ABB RobotStudio station: lab2_v2.rspag

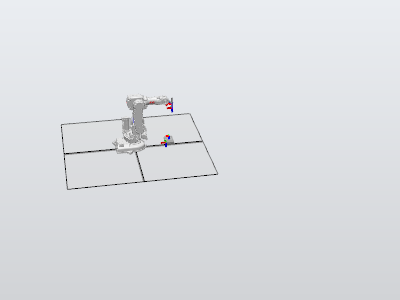
--- station ---
Station lab2_v2 (saved by RobotStudio 25.1.11167.1)
Controller IRB140_6_81
  mechanical unit ROB_1: IRB140T_6_81_C_03, 6 joints, base frame (0, 0, 0) mm
Layout (positions relative to the parent item):
  - IRB140T_6_81_C_03 [mechanism, from %ABB.RobotStudio.Models.IRB140%\IRB140T_6_81_C_G_03.rslib] at (0, 0, 0) mm; joint values [0, 0, 0, 0, 0.5236, 0] (rad or m)
  - marcador [mechanism] at (506.29, 0, 679.5) mm, rotated rx 180 ry 60 rz 180 deg
      TCP punta at (63.25, 0.5, 93.4) mm, rotated rx 0 ry 60 rz 0 deg
      links: Ensamble final v2 (1)
  - WO_LETRAS v4 [part] at (500, 0, 60) mm, rotated rx 0 ry 0 rz -90 deg, size 200 x 120 x 31 mm
Attachment: marcador is attached to IRB140T_6_81_C_03 / Link6

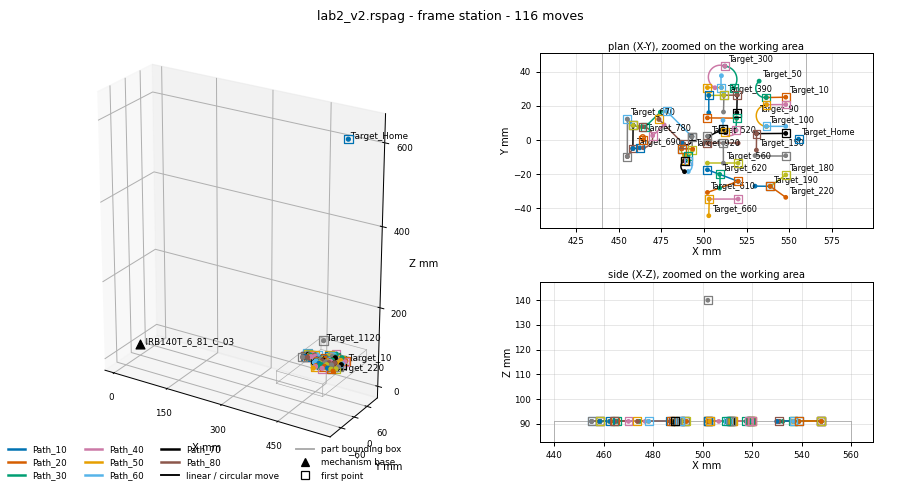
[picture p0: tool path of lab2_v2.rspag in frame station, 116 of 116 moves have a stored position in this frame; points joined in program order, loops and branches not executed]
--- Controller Data/IRB140_6_81/RAPID/TASK1/PROGMOD/CalibData.mod ---
MODULE CalibData
ENDMODULE

--- Controller Data/IRB140_6_81/RAPID/TASK1/PROGMOD/Module1.mod ---
MODULE Module1
        CONST robtarget Target_Home:=[[-115.550957906,100.5,-548.027623724],[1,0,0.000000007,0],[0,-1,0,0],[9E+09,9E+09,9E+09,9E+09,9E+09,9E+09]];
    CONST robtarget Target_10:=[[-108,125.094,-1],[1,0,0,0],[0,0,0,0],[9E+09,9E+09,9E+09,9E+09,9E+09,9E+09]];
    CONST robtarget Target_20:=[[-96.517,124.911,-1],[1,0,0,0],[0,0,0,0],[9E+09,9E+09,9E+09,9E+09,9E+09,9E+09]];
    CONST robtarget Target_30:=[[-96.579,124.938,-1],[1,0,0,0],[0,0,0,0],[9E+09,9E+09,9E+09,9E+09,9E+09,9E+09]];
    CONST robtarget Target_40:=[[-91.246,127.432,-1],[1,0,0,0],[0,0,0,0],[9E+09,9E+09,9E+09,9E+09,9E+09,9E+09]];
    CONST robtarget Target_50:=[[-92.399,134.531,-1],[1,0,0,0],[0,0,0,0],[9E+09,9E+09,9E+09,9E+09,9E+09,9E+09]];
    CONST robtarget Target_60:=[[-108,120.801,-1],[1,0,0,0],[0,0,0,0],[9E+09,9E+09,9E+09,9E+09,9E+09,9E+09]];
    CONST robtarget Target_70:=[[-96.66,120.714,-1],[1,0,0,0],[0,0,0,0],[9E+09,9E+09,9E+09,9E+09,9E+09,9E+09]];
    CONST robtarget Target_80:=[[-96.722,120.654,-1],[1,0,0,0],[0,0,0,0],[9E+09,9E+09,9E+09,9E+09,9E+09,9E+09]];
    CONST robtarget Target_90:=[[-90.707,114.263,-1],[1,0,0,0],[0,0,0,0],[9E+09,9E+09,9E+09,9E+09,9E+09,9E+09]];
    CONST robtarget Target_100:=[[-96.72,107.895,-1],[1,0,0,0],[0,0,0,0],[9E+09,9E+09,9E+09,9E+09,9E+09,9E+09]];
    CONST robtarget Target_110:=[[-96.71,108.02,-1],[1,0,0,0],[0,0,0,0],[9E+09,9E+09,9E+09,9E+09,9E+09,9E+09]];
    CONST robtarget Target_120:=[[-108,108.024,-1],[1,0,0,0],[0,0,0,0],[9E+09,9E+09,9E+09,9E+09,9E+09,9E+09]];
    CONST robtarget Target_130:=[[-108,103.869,-1],[1,0,0,0],[0,0,0,0],[9E+09,9E+09,9E+09,9E+09,9E+09,9E+09]];
    CONST robtarget Target_140:=[[-90.879,103.751,-1],[1,0,0,0],[0,0,0,0],[9E+09,9E+09,9E+09,9E+09,9E+09,9E+09]];
    CONST robtarget Target_150:=[[-90.792,94.077,-1],[1,0,0,0],[0,0,0,0],[9E+09,9E+09,9E+09,9E+09,9E+09,9E+09]];
    CONST robtarget Target_160:=[[-108,90.839,-1],[1,0,0,0],[0,0,0,0],[9E+09,9E+09,9E+09,9E+09,9E+09,9E+09]];
    CONST robtarget Target_170:=[[-90,90.839,-1],[1,0,0,0],[0,0,0,0],[9E+09,9E+09,9E+09,9E+09,9E+09,9E+09]];
    CONST robtarget Target_180:=[[-108,79.52,-1],[1,0,0,0],[0,0,0,0],[9E+09,9E+09,9E+09,9E+09,9E+09,9E+09]];
    CONST robtarget Target_190:=[[-98.899,72.871,-1],[1,0,0,0],[0,0,0,0],[9E+09,9E+09,9E+09,9E+09,9E+09,9E+09]];
    CONST robtarget Target_200:=[[-90,72.954,-1],[1,0,0,0],[0,0,0,0],[9E+09,9E+09,9E+09,9E+09,9E+09,9E+09]];
    CONST robtarget Target_210:=[[-98.899,72.871,-1],[1,0,0,0],[0,0,0,0],[9E+09,9E+09,9E+09,9E+09,9E+09,9E+09]];
    CONST robtarget Target_220:=[[-108,66.388,-1],[1,0,0,0],[0,0,0,0],[9E+09,9E+09,9E+09,9E+09,9E+09,9E+09]];
    CONST robtarget Target_230:=[[-77.51,130.536,-1],[1,0,0,0],[0,0,0,0],[9E+09,9E+09,9E+09,9E+09,9E+09,9E+09]];
    CONST robtarget Target_240:=[[-69.692,143.466,-1],[1,0,0,0],[0,0,0,0],[9E+09,9E+09,9E+09,9E+09,9E+09,9E+09]];
    CONST robtarget Target_250:=[[-67.261,130.559,-1],[1,0,0,0],[0,0,0,0],[9E+09,9E+09,9E+09,9E+09,9E+09,9E+09]];
    CONST robtarget Target_260:=[[-78.123,140.052,-1],[1,0,0,0],[0,0,0,0],[9E+09,9E+09,9E+09,9E+09,9E+09,9E+09]];
    CONST robtarget Target_270:=[[-62.805,137.7,-1],[1,0,0,0],[0,0,0,0],[9E+09,9E+09,9E+09,9E+09,9E+09,9E+09]];
    CONST robtarget Target_280:=[[-77.51,130.536,-1],[1,0,0,0],[0,0,0,0],[9E+09,9E+09,9E+09,9E+09,9E+09,9E+09]];
    CONST robtarget Target_290:=[[-78.383,139.339,-1],[1,0,0,0],[0,0,0,0],[9E+09,9E+09,9E+09,9E+09,9E+09,9E+09]];
    CONST robtarget Target_300:=[[-72.33,143.322,-1],[1,0,0,0],[0,0,0,0],[9E+09,9E+09,9E+09,9E+09,9E+09,9E+09]];
    CONST robtarget Target_310:=[[-72.33,143.322,-1],[1,0,0,0],[0,0,0,0],[9E+09,9E+09,9E+09,9E+09,9E+09,9E+09]];
    CONST robtarget Target_320:=[[-63.095,139.439,-1],[1,0,0,0],[0,0,0,0],[9E+09,9E+09,9E+09,9E+09,9E+09,9E+09]];
    CONST robtarget Target_330:=[[-66.475,130.654,-1],[1,0,0,0],[0,0,0,0],[9E+09,9E+09,9E+09,9E+09,9E+09,9E+09]];
    CONST robtarget Target_340:=[[-62.082,130.754,-1],[1,0,0,0],[0,0,0,0],[9E+09,9E+09,9E+09,9E+09,9E+09,9E+09]];
    CONST robtarget Target_350:=[[-70.29,130.75,-1],[1,0,0,0],[0,0,0,0],[9E+09,9E+09,9E+09,9E+09,9E+09,9E+09]];
    CONST robtarget Target_360:=[[-70.29,137.722,-1],[1,0,0,0],[0,0,0,0],[9E+09,9E+09,9E+09,9E+09,9E+09,9E+09]];
    CONST robtarget Target_370:=[[-79.313,116.071,-1],[1,0,0,0],[0,0,0,0],[9E+09,9E+09,9E+09,9E+09,9E+09,9E+09]];
    CONST robtarget Target_380:=[[-79.514,126.347,-1],[1,0,0,0],[0,0,0,0],[9E+09,9E+09,9E+09,9E+09,9E+09,9E+09]];
    CONST robtarget Target_390:=[[-71.742,126.235,-1],[1,0,0,0],[0,0,0,0],[9E+09,9E+09,9E+09,9E+09,9E+09,9E+09]];
    CONST robtarget Target_400:=[[-71.506,116.416,-1],[1,0,0,0],[0,0,0,0],[9E+09,9E+09,9E+09,9E+09,9E+09,9E+09]];
    CONST robtarget Target_410:=[[-71.721,126.247,-1],[1,0,0,0],[0,0,0,0],[9E+09,9E+09,9E+09,9E+09,9E+09,9E+09]];
    CONST robtarget Target_420:=[[-62.895,126.149,-1],[1,0,0,0],[0,0,0,0],[9E+09,9E+09,9E+09,9E+09,9E+09,9E+09]];
    CONST robtarget Target_430:=[[-62.874,116.003,-1],[1,0,0,0],[0,0,0,0],[9E+09,9E+09,9E+09,9E+09,9E+09,9E+09]];
    CONST robtarget Target_440:=[[-62.082,112.96,-1],[1,0,0,0],[0,0,0,0],[9E+09,9E+09,9E+09,9E+09,9E+09,9E+09]];
    CONST robtarget Target_450:=[[-79.192,112.835,-1],[1,0,0,0],[0,0,0,0],[9E+09,9E+09,9E+09,9E+09,9E+09,9E+09]];
    CONST robtarget Target_460:=[[-78.805,105.664,-1],[1,0,0,0],[0,0,0,0],[9E+09,9E+09,9E+09,9E+09,9E+09,9E+09]];
    CONST robtarget Target_470:=[[-75.79,102.587,-1],[1,0,0,0],[0,0,0,0],[9E+09,9E+09,9E+09,9E+09,9E+09,9E+09]];
    CONST robtarget Target_480:=[[-72.357,104.51,-1],[1,0,0,0],[0,0,0,0],[9E+09,9E+09,9E+09,9E+09,9E+09,9E+09]];
    CONST robtarget Target_490:=[[-71.207,106.55,-1],[1,0,0,0],[0,0,0,0],[9E+09,9E+09,9E+09,9E+09,9E+09,9E+09]];
    CONST robtarget Target_500:=[[-71.216,111.54,-1],[1,0,0,0],[0,0,0,0],[9E+09,9E+09,9E+09,9E+09,9E+09,9E+09]];
    CONST robtarget Target_510:=[[-71.224,106.472,-1],[1,0,0,0],[0,0,0,0],[9E+09,9E+09,9E+09,9E+09,9E+09,9E+09]];
    CONST robtarget Target_520:=[[-62.667,102.098,-1],[1,0,0,0],[0,0,0,0],[9E+09,9E+09,9E+09,9E+09,9E+09,9E+09]];
    CONST robtarget Target_530:=[[-62.082,98.14,-1],[1,0,0,0],[0,0,0,0],[9E+09,9E+09,9E+09,9E+09,9E+09,9E+09]];
    CONST robtarget Target_540:=[[-80.082,98.14,-1],[1,0,0,0],[0,0,0,0],[9E+09,9E+09,9E+09,9E+09,9E+09,9E+09]];
    CONST robtarget Target_550:=[[-71.397,98.148,-1],[1,0,0,0],[0,0,0,0],[9E+09,9E+09,9E+09,9E+09,9E+09,9E+09]];
    CONST robtarget Target_560:=[[-71.446,86.432,-1],[1,0,0,0],[0,0,0,0],[9E+09,9E+09,9E+09,9E+09,9E+09,9E+09]];
    CONST robtarget Target_570:=[[-80.082,86.454,-1],[1,0,0,0],[0,0,0,0],[9E+09,9E+09,9E+09,9E+09,9E+09,9E+09]];
    CONST robtarget Target_580:=[[-62.082,86.454,-1],[1,0,0,0],[0,0,0,0],[9E+09,9E+09,9E+09,9E+09,9E+09,9E+09]];
    CONST robtarget Target_590:=[[-62.082,82.562,-1],[1,0,0,0],[0,0,0,0],[9E+09,9E+09,9E+09,9E+09,9E+09,9E+09]];
    CONST robtarget Target_600:=[[-80.082,75.79,-1],[1,0,0,0],[0,0,0,0],[9E+09,9E+09,9E+09,9E+09,9E+09,9E+09]];
    CONST robtarget Target_610:=[[-62.082,69.258,-1],[1,0,0,0],[0,0,0,0],[9E+09,9E+09,9E+09,9E+09,9E+09,9E+09]];
    CONST robtarget Target_620:=[[-69.26,79.86,-1],[1,0,0,0],[0,0,0,0],[9E+09,9E+09,9E+09,9E+09,9E+09,9E+09]];
    CONST robtarget Target_630:=[[-69.26,71.805,-1],[1,0,0,0],[0,0,0,0],[9E+09,9E+09,9E+09,9E+09,9E+09,9E+09]];
    CONST robtarget Target_640:=[[-80.082,65.389,-1],[1,0,0,0],[0,0,0,0],[9E+09,9E+09,9E+09,9E+09,9E+09,9E+09]];
    CONST robtarget Target_650:=[[-63.123,65.37,-1],[1,0,0,0],[0,0,0,0],[9E+09,9E+09,9E+09,9E+09,9E+09,9E+09]];
    CONST robtarget Target_660:=[[-62.874,55.597,-1],[1,0,0,0],[0,0,0,0],[9E+09,9E+09,9E+09,9E+09,9E+09,9E+09]];
    CONST robtarget Target_670:=[[-15.067,112.238,-1],[1,0,0,0],[0,0,0,0],[9E+09,9E+09,9E+09,9E+09,9E+09,9E+09]];
    CONST robtarget Target_680:=[[-18.49,108.612,-1],[1,0,0,0],[0,0,0,0],[9E+09,9E+09,9E+09,9E+09,9E+09,9E+09]];
    CONST robtarget Target_690:=[[-18.364,95.026,-1],[1,0,0,0],[0,0,0,0],[9E+09,9E+09,9E+09,9E+09,9E+09,9E+09]];
    CONST robtarget Target_700:=[[-15.102,90.307,-1],[1,0,0,0],[0,0,0,0],[9E+09,9E+09,9E+09,9E+09,9E+09,9E+09]];
    CONST robtarget Target_710:=[[-15.158,112.207,-1],[1,0,0,0],[0,0,0,0],[9E+09,9E+09,9E+09,9E+09,9E+09,9E+09]];
    CONST robtarget Target_720:=[[-18.49,108.612,-1],[1,0,0,0],[0,0,0,0],[9E+09,9E+09,9E+09,9E+09,9E+09,9E+09]];
    CONST robtarget Target_730:=[[-22.178,107.545,-1],[1,0,0,0],[0,0,0,0],[9E+09,9E+09,9E+09,9E+09,9E+09,9E+09]];
    CONST robtarget Target_740:=[[-29.789,101.463,-1],[1,0,0,0],[0,0,0,0],[9E+09,9E+09,9E+09,9E+09,9E+09,9E+09]];
    CONST robtarget Target_750:=[[-22.386,95.374,-1],[1,0,0,0],[0,0,0,0],[9E+09,9E+09,9E+09,9E+09,9E+09,9E+09]];
    CONST robtarget Target_760:=[[-18.397,95.013,-1],[1,0,0,0],[0,0,0,0],[9E+09,9E+09,9E+09,9E+09,9E+09,9E+09]];
    CONST robtarget Target_770:=[[-24.444,100.113,-1],[1,0,0,0],[0,0,0,0],[9E+09,9E+09,9E+09,9E+09,9E+09,9E+09]];
    CONST robtarget Target_780:=[[-24.359,103.047,-1],[1,0,0,0],[0,0,0,0],[9E+09,9E+09,9E+09,9E+09,9E+09,9E+09]];
    CONST robtarget Target_790:=[[-24.554,100.141,-1],[1,0,0,0],[0,0,0,0],[9E+09,9E+09,9E+09,9E+09,9E+09,9E+09]];
    CONST robtarget Target_800:=[[-25.496,107.635,-1],[1,0,0,0],[0,0,0,0],[9E+09,9E+09,9E+09,9E+09,9E+09,9E+09]];
    CONST robtarget Target_810:=[[-34.48,116.37,-1],[1,0,0,0],[0,0,0,0],[9E+09,9E+09,9E+09,9E+09,9E+09,9E+09]];
    CONST robtarget Target_820:=[[-29.986,102.575,-1],[1,0,0,0],[0,0,0,0],[9E+09,9E+09,9E+09,9E+09,9E+09,9E+09]];
    CONST robtarget Target_830:=[[-36.719,108.862,-1],[1,0,0,0],[0,0,0,0],[9E+09,9E+09,9E+09,9E+09,9E+09,9E+09]];
    CONST robtarget Target_840:=[[-33.544,112.115,-1],[1,0,0,0],[0,0,0,0],[9E+09,9E+09,9E+09,9E+09,9E+09,9E+09]];
    CONST robtarget Target_850:=[[-34.336,116.216,-1],[1,0,0,0],[0,0,0,0],[9E+09,9E+09,9E+09,9E+09,9E+09,9E+09]];
    CONST robtarget Target_860:=[[-38.148,116.925,-1],[1,0,0,0],[0,0,0,0],[9E+09,9E+09,9E+09,9E+09,9E+09,9E+09]];
    CONST robtarget Target_870:=[[-52.946,102.081,-1],[1,0,0,0],[0,0,0,0],[9E+09,9E+09,9E+09,9E+09,9E+09,9E+09]];
    CONST robtarget Target_880:=[[-52.107,98.145,-1],[1,0,0,0],[0,0,0,0],[9E+09,9E+09,9E+09,9E+09,9E+09,9E+09]];
    CONST robtarget Target_890:=[[-48.099,97.619,-1],[1,0,0,0],[0,0,0,0],[9E+09,9E+09,9E+09,9E+09,9E+09,9E+09]];
    CONST robtarget Target_900:=[[-33.658,112.146,-1],[1,0,0,0],[0,0,0,0],[9E+09,9E+09,9E+09,9E+09,9E+09,9E+09]];
    CONST robtarget Target_910:=[[-52.993,101.964,-1],[1,0,0,0],[0,0,0,0],[9E+09,9E+09,9E+09,9E+09,9E+09,9E+09]];
    CONST robtarget Target_920:=[[-53.234,94.103,-1],[1,0,0,0],[0,0,0,0],[9E+09,9E+09,9E+09,9E+09,9E+09,9E+09]];
    CONST robtarget Target_930:=[[-50.381,90.681,-1],[1,0,0,0],[0,0,0,0],[9E+09,9E+09,9E+09,9E+09,9E+09,9E+09]];
    CONST robtarget Target_940:=[[-46.922,94.871,-1],[1,0,0,0],[0,0,0,0],[9E+09,9E+09,9E+09,9E+09,9E+09,9E+09]];
    CONST robtarget Target_950:=[[-47.013,98.691,-1],[1,0,0,0],[0,0,0,0],[9E+09,9E+09,9E+09,9E+09,9E+09,9E+09]];
    CONST robtarget Target_960:=[[-47.015,94.837,-1],[1,0,0,0],[0,0,0,0],[9E+09,9E+09,9E+09,9E+09,9E+09,9E+09]];
    CONST robtarget Target_970:=[[-53.429,94.778,-1],[1,0,0,0],[0,0,0,0],[9E+09,9E+09,9E+09,9E+09,9E+09,9E+09]];
    CONST robtarget Target_980:=[[-50.711,90.745,-1],[1,0,0,0],[0,0,0,0],[9E+09,9E+09,9E+09,9E+09,9E+09,9E+09]];
    CONST robtarget Target_990:=[[-50.919,87.918,-1],[1,0,0,0],[0,0,0,0],[9E+09,9E+09,9E+09,9E+09,9E+09,9E+09]];
    CONST robtarget Target_1000:=[[-49.871,86.938,-1],[1,0,0,0],[0,0,0,0],[9E+09,9E+09,9E+09,9E+09,9E+09,9E+09]];
    CONST robtarget Target_1010:=[[-48.634,87.988,-1],[1,0,0,0],[0,0,0,0],[9E+09,9E+09,9E+09,9E+09,9E+09,9E+09]];
    CONST robtarget Target_1020:=[[-48.643,90.985,-1],[1,0,0,0],[0,0,0,0],[9E+09,9E+09,9E+09,9E+09,9E+09,9E+09]];
    CONST robtarget Target_1030:=[[-50.973,87.895,-1],[1,0,0,0],[0,0,0,0],[9E+09,9E+09,9E+09,9E+09,9E+09,9E+09]];
    CONST robtarget Target_1040:=[[-53.036,84.502,-1],[1,0,0,0],[0,0,0,0],[9E+09,9E+09,9E+09,9E+09,9E+09,9E+09]];
    CONST robtarget Target_1050:=[[-50.844,81.528,-1],[1,0,0,0],[0,0,0,0],[9E+09,9E+09,9E+09,9E+09,9E+09,9E+09]];
    CONST robtarget Target_1060:=[[-48.691,87.835,-1],[1,0,0,0],[0,0,0,0],[9E+09,9E+09,9E+09,9E+09,9E+09,9E+09]];
    CONST robtarget Target_1070:=[[-46.541,84.777,-1],[1,0,0,0],[0,0,0,0],[9E+09,9E+09,9E+09,9E+09,9E+09,9E+09]];
    CONST robtarget Target_1080:=[[-48.635,81.464,0],[1,0,0,0],[0,0,0,0],[9E+09,9E+09,9E+09,9E+09,9E+09,9E+09]];
    CONST robtarget Target_1090:=[[-24.027,107.791,-1],[1,0,0,0],[0,0,0,0],[9E+09,9E+09,9E+09,9E+09,9E+09,9E+09]];
    CONST robtarget Target_1100:=[[-29.971,101.827,-1],[1,0,0,0],[0,0,0,0],[9E+09,9E+09,9E+09,9E+09,9E+09,9E+09]];
    CONST robtarget Target_1110:=[[-24.506,95.448,-1],[1,0,0,0],[0,0,0,0],[9E+09,9E+09,9E+09,9E+09,9E+09,9E+09]];
    CONST robtarget Target_1120:=[[-62.082,102.239,-50],[1,0,0,0],[0,0,0,0],[9E+09,9E+09,9E+09,9E+09,9E+09,9E+09]];
    PERS tooldata punta:=[TRUE,[[63.248,0.5,93.396],[0.866025404,0,0.5,0]],[1,[0,0,1],[1,0,0,0],0,0,0]];
    TASK PERS wobjdata Workobject_2:=[FALSE,TRUE,"",[[0,0,60],[1,0,0,0]],[[440,-100,30],[0,0,1,0]]];
!***********************************************************
    !
    ! M?dulo:  Module1
    !
    ! Descripción:
    !   <Introduzca la descripción aquí>
    !
    ! Autor: MacBook Air
    !
    ! Versión: 1.0
    !
    !***********************************************************


    !***********************************************************
    !
    ! Procedimiento Main
    !
    !   Este es el punto de entrada de su programa
    !
    !***********************************************************
    PROC main()
        Path_10;
        Path_600;
        Path_20;
        Path_30;
        Path_600;
        Path_40;
        Path_50;
        Path_60;
        Path_600;
        Path_70;
        Path_80;
        Path_600;
        Path_90;
        Path_600;
        Path_100;
        Path_110;
        Path_120;
        Path_600;
        Path_130;
        Path_140;
        Path_150;
        Path_160;
        Path_600;
        Path_170;
        Path_180;
        Path_190;
        Path_200;
        Path_210;
        Path_600;
        Path_220;
        Path_230;
        Path_240;
        Path_250;
        Path_260;
        Path_270;
        Path_600;
        Path_280;
        Path_290;
        Path_300;
        Path_600;
        Path_310;
        Path_320;
        Path_330;
        Path_600;
        Path_340;
        Path_350;
        Path_600;
        Path_360;
        Path_370;
        Path_380;
        Path_390;
        Path_600;
        Path_400;
        Path_600;
        Path_420;
        Path_600;
        Path_440;
        Path_600;
        Path_450;
        Path_600;
        Path_460;
        Path_470;
        Path_480;
        Path_490;
        Path_600;
        Path_500;
        Path_510;
        Path_520;
        Path_600;
        Path_530;
        Path_600;
        Path_540;
        Path_550;
        Path_560;
        Path_600;
        Path_570;
        Path_580;
        Path_600;
        Path_590;
        Path_600;
        Path_10;



    ENDPROC
    PROC Path_10()
        MoveJ Target_Home,v100,z10,punta\WObj:=Workobject_2;
    ENDPROC
    PROC Path_20()
        MoveJ Target_10,v100,z10,punta\WObj:=Workobject_2;
        MoveL Target_20,v100,z10,punta\WObj:=Workobject_2;
    ENDPROC
    PROC Path_30()
        MoveJ Target_30,v100,z10,punta\WObj:=Workobject_2;
        MoveC Target_40,Target_50,v100,z10,punta\WObj:=Workobject_2;
    ENDPROC
    PROC Path_40()
        MoveJ Target_60,v100,z10,punta\WObj:=Workobject_2;
        MoveL Target_70,v100,z10,punta\WObj:=Workobject_2;
    ENDPROC
    PROC Path_50()
        MoveJ Target_80,v100,z10,punta\WObj:=Workobject_2;
        MoveC Target_90,Target_100,v1000,z100,punta\WObj:=Workobject_2;
    ENDPROC
    PROC Path_60()
        MoveJ Target_110,v100,z10,punta\WObj:=Workobject_2;
        MoveL Target_120,v100,z10,punta\WObj:=Workobject_2;
    ENDPROC
    PROC Path_70()
        MoveJ Target_130,v100,z10,punta\WObj:=Workobject_2;
        MoveL Target_140,v100,z10,punta\WObj:=Workobject_2;
    ENDPROC
    PROC Path_80()
        MoveJ Target_140,v100,z10,punta\WObj:=Workobject_2;
        MoveL Target_150,v100,z10,punta\WObj:=Workobject_2;
    ENDPROC
    PROC Path_90()
        MoveJ Target_160,v100,z10,punta\WObj:=Workobject_2;
        MoveL Target_170,v100,z10,punta\WObj:=Workobject_2;
    ENDPROC
    PROC Path_100()
        MoveJ Target_180,v100,z10,punta\WObj:=Workobject_2;
        MoveL Target_190,v100,z10,punta\WObj:=Workobject_2;
    ENDPROC
    PROC Path_110()
        MoveJ Target_190,v100,z10,punta\WObj:=Workobject_2;
        MoveL Target_200,v100,z10,punta\WObj:=Workobject_2;
    ENDPROC
    PROC Path_120()
        MoveJ Target_210,v100,z10,punta\WObj:=Workobject_2;
        MoveL Target_220,v100,z10,punta\WObj:=Workobject_2;
    ENDPROC
    PROC Path_130()
        MoveJ Target_280,v100,z10,punta\WObj:=Workobject_2;
        MoveC Target_290,Target_300,v100,z10,punta\WObj:=Workobject_2;
    ENDPROC
    PROC Path_140()
        MoveJ Target_310,v100,z10,punta\WObj:=Workobject_2;
        MoveC Target_320,Target_330,v100,z10,punta\WObj:=Workobject_2;

    ENDPROC
    PROC Path_150()
        MoveJ Target_340,v100,z10,punta\WObj:=Workobject_2;
        MoveL Target_350,v100,z10,punta\WObj:=Workobject_2;
    ENDPROC
    PROC Path_160()
        MoveJ Target_350,v100,z10,punta\WObj:=Workobject_2;
        MoveL Target_360,v100,z10,punta\WObj:=Workobject_2;
    ENDPROC
    PROC Path_170()
        MoveJ Target_370,v100,z10,punta\WObj:=Workobject_2;
        MoveL Target_380,v100,z10,punta\WObj:=Workobject_2;
    ENDPROC
    PROC Path_180()
        MoveJ Target_380,v100,z10,punta\WObj:=Workobject_2;
        MoveL Target_390,v100,z10,punta\WObj:=Workobject_2;
    ENDPROC
    PROC Path_190()
        MoveJ Target_390,v100,z10,punta\WObj:=Workobject_2;
        MoveL Target_400,v100,z10,punta\WObj:=Workobject_2;
    ENDPROC
    PROC Path_200()
        MoveJ Target_410,v100,z10,punta\WObj:=Workobject_2;
        MoveL Target_420,v100,z10,punta\WObj:=Workobject_2;
    ENDPROC
    PROC Path_210()
        MoveJ Target_420,v100,z10,punta\WObj:=Workobject_2;
        MoveL Target_430,v100,z10,punta\WObj:=Workobject_2;
    ENDPROC
    PROC Path_220()
        MoveJ Target_440,v100,z10,punta\WObj:=Workobject_2;
        MoveL Target_450,v100,z10,punta\WObj:=Workobject_2;
    ENDPROC
    PROC Path_230()
        MoveJ Target_450,v100,z10,punta\WObj:=Workobject_2;
        MoveL Target_460,v100,z10,punta\WObj:=Workobject_2;
    ENDPROC
    PROC Path_240()
        MoveJ Target_460,v100,z10,punta\WObj:=Workobject_2;
        MoveC Target_470,Target_480,v100,z10,punta\WObj:=Workobject_2;

    ENDPROC
    PROC Path_250()
        MoveJ Target_480,v100,z10,punta\WObj:=Workobject_2;
        MoveL Target_490,v100,z10,punta\WObj:=Workobject_2;
    ENDPROC
    PROC Path_260()
        MoveJ Target_490,v100,z10,punta\WObj:=Workobject_2;
        MoveL Target_500,v100,z10,punta\WObj:=Workobject_2;
    ENDPROC
    PROC Path_270()
        MoveJ Target_510,v100,z10,punta\WObj:=Workobject_2;
        MoveL Target_520,v100,z10,punta\WObj:=Workobject_2;
    ENDPROC
    PROC Path_280()
        MoveJ Target_530,v100,z10,punta\WObj:=Workobject_2;
        MoveL Target_540,v100,z10,punta\WObj:=Workobject_2;
    ENDPROC
    PROC Path_290()
        MoveJ Target_550,v100,z10,punta\WObj:=Workobject_2;
        MoveL Target_560,v100,z10,punta\WObj:=Workobject_2;
    ENDPROC
    PROC Path_300()
        MoveJ Target_570,v100,z10,punta\WObj:=Workobject_2;
        MoveL Target_580,v100,z10,punta\WObj:=Workobject_2;
    ENDPROC
    PROC Path_310()
        MoveJ Target_590,v100,z10,punta\WObj:=Workobject_2;
        MoveL Target_600,v100,z10,punta\WObj:=Workobject_2;
    ENDPROC
    PROC Path_320()
        MoveJ Target_600,v100,z10,punta\WObj:=Workobject_2;
        MoveL Target_610,v100,z10,punta\WObj:=Workobject_2;
    ENDPROC
    PROC Path_330()
        MoveJ Target_620,v100,z10,punta\WObj:=Workobject_2;
        MoveL Target_630,v100,z10,punta\WObj:=Workobject_2;
    ENDPROC
    PROC Path_340()
        MoveJ Target_640,v100,z10,punta\WObj:=Workobject_2;
        MoveL Target_650,v100,z10,punta\WObj:=Workobject_2;
    ENDPROC
    PROC Path_350()
        MoveJ Target_650,v100,z10,punta\WObj:=Workobject_2;
        MoveL Target_660,v100,z10,punta\WObj:=Workobject_2;
    ENDPROC
    PROC Path_360()
        MoveJ Target_670,v100,z10,punta\WObj:=Workobject_2;
        MoveL Target_680,v100,z10,punta\WObj:=Workobject_2;
    ENDPROC
    PROC Path_370()
        MoveJ Target_680,v100,z10,punta\WObj:=Workobject_2;
        MoveL Target_690,v100,z10,punta\WObj:=Workobject_2;
    ENDPROC
    PROC Path_380()
        MoveJ Target_690,v100,z10,punta\WObj:=Workobject_2;
        MoveL Target_700,v100,z10,punta\WObj:=Workobject_2;
    ENDPROC
    PROC Path_390()
        MoveJ Target_700,v1000,z10,punta\WObj:=Workobject_2;
        MoveL Target_710,v1000,z10,punta\WObj:=Workobject_2;
    ENDPROC
    PROC Path_400()
        MoveJ Target_720,v100,z10,punta\WObj:=Workobject_2;
        MoveL Target_730,v100,z10,punta\WObj:=Workobject_2;
    ENDPROC

    PROC Path_420()
        MoveJ Target_750,v100,z10,punta\WObj:=Workobject_2;
        MoveL Target_760,v100,z10,punta\WObj:=Workobject_2;
    ENDPROC
    PROC Path_430()
        MoveJ Target_770,v100,z10,punta\WObj:=Workobject_2;
        MoveC Target_780,Target_790,v100,z10,punta\WObj:=Workobject_2;

    ENDPROC
    PROC Path_440()
        MoveJ Target_800,v100,z10,punta\WObj:=Workobject_2;
        MoveL Target_810,v100,z10,punta\WObj:=Workobject_2;
    ENDPROC
    PROC Path_450()
        MoveJ Target_820,v100,z10,punta\WObj:=Workobject_2;
        MoveL Target_830,v100,z10,punta\WObj:=Workobject_2;
    ENDPROC
    PROC Path_460()
        MoveJ Target_840,v100,z10,punta\WObj:=Workobject_2;
        MoveC Target_850,Target_860,v100,z10,punta\WObj:=Workobject_2;
    ENDPROC
    PROC Path_470()
        MoveJ Target_860,v100,z10,punta\WObj:=Workobject_2;
        MoveL Target_870,v100,z10,punta\WObj:=Workobject_2;
    ENDPROC
    PROC Path_480()
        MoveJ Target_870,v100,z10,punta\WObj:=Workobject_2;
        MoveC Target_880,Target_890,v100,z10,punta\WObj:=Workobject_2;
    ENDPROC
    PROC Path_490()
        MoveJ Target_890,v100,z10,punta\WObj:=Workobject_2;
        MoveL Target_900,v100,z10,punta\WObj:=Workobject_2;
    ENDPROC
    PROC Path_500()
        MoveJ Target_910,v100,z10,punta\WObj:=Workobject_2;
        MoveL Target_920,v100,z10,punta\WObj:=Workobject_2;
    ENDPROC
    PROC Path_510()
        MoveJ Target_920,v100,z10,punta\WObj:=Workobject_2;
        MoveC Target_930,Target_940,v100,z10,punta\WObj:=Workobject_2;
    ENDPROC
    PROC Path_520()
        MoveJ Target_940,v100,z10,punta\WObj:=Workobject_2;
        MoveL Target_950,v100,z10,punta\WObj:=Workobject_2;
    ENDPROC
    PROC Path_530()
        MoveJ Target_960,v100,z10,punta\WObj:=Workobject_2;
        MoveL Target_970,v100,z10,punta\WObj:=Workobject_2;
    ENDPROC
    PROC Path_540()
        MoveJ Target_980,v100,z10,punta\WObj:=Workobject_2;
        MoveL Target_990,v100,z10,punta\WObj:=Workobject_2;
    ENDPROC
    PROC Path_550()
        MoveJ Target_990,v100,z10,punta\WObj:=Workobject_2;
        MoveC Target_1000,Target_1010,v100,z10,punta\WObj:=Workobject_2;

    ENDPROC
    PROC Path_560()
        MoveJ Target_1010,v100,z10,punta\WObj:=Workobject_2;
        MoveL Target_1020,v100,z10,punta\WObj:=Workobject_2;
    ENDPROC
    PROC Path_570()
        MoveJ Target_1030,v100,z10,punta\WObj:=Workobject_2;
        MoveC Target_1040,Target_1050,v100,z10,punta\WObj:=Workobject_2;

    ENDPROC
    PROC Path_580()
        MoveJ Target_1060,v100,z10,punta\WObj:=Workobject_2;
        MoveC Target_1070,Target_1080,v100,z10,punta\WObj:=Workobject_2;

    ENDPROC
    PROC Path_590()
        MoveJ Target_1090,v100,z10,punta\WObj:=Workobject_2;
        MoveC Target_1100,Target_1110,v100,z10,punta\WObj:=Workobject_2;

    ENDPROC
    PROC Path_600()
        MoveJ Target_1120,v100,z10,punta\WObj:=Workobject_2;
    ENDPROC
ENDMODULE
